// TIA Portal V20 export
DATA_BLOCK "LPFE_RecordBuffer"   // DB244
TITLE = Buffer of RequestOrderInfo messages
// Buffer to store record messages (7,8) until distributed
// stored: Access Published, MemoryReserve 100, Namespace PFE
   VAR
      buffer { ExternalAccessible := 'False'; ExternalVisible := 'False'; ExternalWritable := 'False'} : Array[0.._.LE_NUMBER_MESSAGES_RECORD_BUFFER] of "LPFE_typePFEDataReqEnvelope";   // Buffer where record messages are written and read
      mgmtBuffer { ExternalAccessible := 'False'; ExternalVisible := 'False'; ExternalWritable := 'False'} : "LPFE_typeMsgBuffer";   // Management Structure of buffer
      currentCriticalRecord { ExternalAccessible := 'False'; ExternalVisible := 'False'; ExternalWritable := 'False'} : "LPFE_typeCriticalRecEnvelope";
   END_VAR
BEGIN
   // currentCriticalRecord.waitingForCriticalAck : TRUE: Critical Acknowledge required for special events
END_DATA_BLOCK
